{attribute 'GeneratedUsingTerminal: EL6851-0000-0017'}
{attribute addProperty BoxType "EL6851-0000-0017"}
{attribute addProperty Id "EtcSlaveTerminalBaseDMX_StatusAT %I*DMX_Status_5716F9AF9DMX_ControlAT %Q*DMX_Control_8D35CC316DMX_Channel_1_64AT %Q*DMX_Channel_FF1F0CB664DMX_Channel_65_128AT %Q*DMX_Channel_DC7E303664DMX_Channel_129_192AT %Q*DMX_Channel_60D8A7A564DMX_Channel_193_256AT %Q*DMX_Channel_AEBD222664DMX_Channel_257_320AT %Q*DMX_Channel_346A633C64DMX_Channel_321_384AT %Q*DMX_Channel_C9FE109C64DMX_Channel_385_448AT %Q*DMX_Channel_A44FB6B664DMX_Channel_449_512AT %Q*DMX_Channel_BD63FDF664WcStateAT %I*WcState_9091E0EB2InfoDataAT %I*InfoData_32EB74EA10"}
{attribute addProperty CRC "2842761291"}
{attribute addProperty Size "539"}
TYPE EL6851_A971184B EXTENDS EtcSlaveTerminalBase :
STRUCT
	{attribute addProperty Name "DMX_Status"}
	DMX_Status : DMX_Status_5716F9AF;
	{attribute addProperty Name "DMX_Control"}
	DMX_Control : DMX_Control_8D35CC31;
	{attribute addProperty Name "DMX_Channel_1_64"}
	DMX_Channel_1_64 : DMX_Channel_FF1F0CB6;
	{attribute addProperty Name "DMX_Channel_65_128"}
	DMX_Channel_65_128 : DMX_Channel_DC7E3036;
	{attribute addProperty Name "DMX_Channel_129_192"}
	DMX_Channel_129_192 : DMX_Channel_60D8A7A5;
	{attribute addProperty Name "DMX_Channel_193_256"}
	DMX_Channel_193_256 : DMX_Channel_AEBD2226;
	{attribute addProperty Name "DMX_Channel_257_320"}
	DMX_Channel_257_320 : DMX_Channel_346A633C;
	{attribute addProperty Name "DMX_Channel_321_384"}
	DMX_Channel_321_384 : DMX_Channel_C9FE109C;
	{attribute addProperty Name "DMX_Channel_385_448"}
	DMX_Channel_385_448 : DMX_Channel_A44FB6B6;
	{attribute addProperty Name "DMX_Channel_449_512"}
	DMX_Channel_449_512 : DMX_Channel_BD63FDF6;
	{attribute addProperty Name "WcState"}
	WcState : WcState_9091E0EB;
	{attribute addProperty Name "InfoData"}
	InfoData : InfoData_32EB74EA;
END_STRUCT
END_TYPE

(* stored: Version 1.2.0.0, ProductVersion 3.1.4024.9
   DUT EL6851_A971184B: Id {91b9b9f4-505d-410f-9543-14a31107d1f8} *)
